{attribute addProperty BoxType "EL5151-0000-0017"}
{attribute addProperty Id "ENC_InputsAT %I*ENC_Inputs_B13A87D6144180ENC_Inputs_1AT %I*ENC_Inputs_AC51B8A03240ENC_OutputsAT %Q*ENC_Outputs_90374C536480WcStateAT %I*WcState_98A4DF7520.250InfoDataAT %I*InfoData_BC63D37F80100"}
{attribute addProperty CRC "2541834964"}
{attribute addProperty SizeInBites "322"}
{attribute addProperty SizeInBytes "40.25"}
TYPE EL5151_023DC4F2 :
STRUCT
	{attribute addProperty Name "ENC_Inputs"}
	ENC_Inputs : ENC_Inputs_B13A87D6;
	{attribute addProperty Name "ENC_Inputs_1"}
	ENC_Inputs_1 : ENC_Inputs_AC51B8A0;
	{attribute addProperty Name "ENC_Outputs"}
	ENC_Outputs : ENC_Outputs_90374C53;
	{attribute addProperty Name "WcState"}
	WcState : WcState_98A4DF75;
	{attribute addProperty Name "InfoData"}
	InfoData : InfoData_BC63D37F;
END_STRUCT
END_TYPE

(* stored: Version 1.2.0.0, ProductVersion 3.1.4024.9
   DUT EL5151_023DC4F2: Id {6140c793-56c2-4edc-b1d4-a3324160ea1f} *)
